{attribute 'qualified_only'}
VAR_GLOBAL
	
myPlcAppSystemInfo:PlcAppSystemInfo;
myPlcInfoTask1 : PlcTaskSystemInfo;
myPlcInfoTask2 : PlcTaskSystemInfo;
myPlcInfoTask3 : PlcTaskSystemInfo;
myPlcInfoTask4 : PlcTaskSystemInfo;
myPlcInfoTask5 : PlcTaskSystemInfo;
myPlcInfoTask6 : PlcTaskSystemInfo;


ScanTimeReq:REAL; //the programmed task scan time, e.g. 1, 10, 15, 30ms, etc
ScanTimeAct:REAL; //the last scan time, effective current scan time.

ScanTimeRecord:REAL; //the record scan time
ScanTimeRecordScan:LREAL; //the scan number of the record scan time


//EtherCAT masters mapped into all memory
ecMasterData :ARRAY[1..etherCATdiag.maxNumEtherCATmasters] OF typeEtherCATmasters;

thetime: TIMESTRUCT;

oneMilliSecond: BOOL;
hundredMilliSecond:BOOL;
OneSecond: BOOL;
TwoSecond: BOOL;
TenSecond: BOOL;

StartPulse:BOOL;

PulseOneMilliSecond: BOOL;
PulseHundredMilliSecond:BOOL;
PulseOneSecond: BOOL;
PulseTwoSecond: BOOL;
PulseTenSecond: BOOL;

timeDT: DT;

gSetup:typeSetupMachine; //setup data for machine

cpuusageval:UDINT; //CPU usage in percent

symCount: UDINT; //Max. number of available symbols 
sysSize: UDINT; //Max. byte size of symbol information

LatencyMicroSec:UDINT;	//Actual latency in µs 
MaxLatencyMicroSec:UDINT; //Maximum latency in µs

TCRestartReq:BOOL; //restart TC
TCStopReq:BOOL; //stop TC
TCConfigReq:BOOL; //stop TC
NThostname:T_MaxString; //NT hostname
networkadaptors: ARRAY [0..MAX_LOCAL_ADAPTERS] OF ST_IpAdapterInfo;

sysDeviceInfo: Tc2_Utilities.ST_DeviceIdentificationEx;
sysDeviceUpdate:BOOL;

AmsNetIdstr: STRING(23);
AmsNetIdbytes: ARRAY[0..5] OF BYTE;

gHappyBirthday:BOOL;


END_VAR

(* stored: Version 1.1.0.1, ProductVersion 3.1.4024.11
   GVL System: Id {fa1ba82a-a43b-47a5-9097-4bd33bbfce0d} *)
